FUNCTION_BLOCK EcMasterFrameCount IMPLEMENTS IEcTask
VAR_INPUT
END_VAR
VAR_OUTPUT
END_VAR
VAR
	iState : INT;
	masterFrameCount : Tc2_EtherCAT.FB_EcMasterFrameCount;
	_execute: BOOL;
	_done: BOOL;
	_busy: BOOL;
	_error: BOOL;
	_netId: AMSNETID;
END_VAR

CASE iState OF
	0:
		IF _execute THEN
			_done := FALSE;
			_busy := TRUE;
			_error := FALSE;
			masterFrameCount.bExecute := TRUE;
			IF masterFrameCount.bBusy THEN
				iState := 10;
				_execute := false;
			END_IF
		END_IF
	10:
		IF NOT masterFrameCount.bBusy THEN
			IF NOT masterFrameCount.bError THEN
				_done := TRUE;
			ELSE
				_error := TRUE;
			END_IF
			_busy := FALSE;
			masterFrameCount.bExecute := FALSE;
			iState := 0;
		END_IF
END_CASE

masterFrameCount(sNetId := Tc2_System.F_CreateAmsNetId(nIds := NetId));

{warning 'add method implementation '}
METHOD Abort : BOOL
masterFrameCount.bExecute := FALSE;
_busy := FALSE;
_execute := FALSE;
Abort := TRUE;
iState := 0;
END_METHOD

{warning 'add property implementation'}
PROPERTY Busy : BOOL
GET
Busy := _busy;
END_GET
END_PROPERTY

{warning 'add property implementation'}
PROPERTY Done : BOOL
GET
Done := _done;
END_GET
END_PROPERTY

{warning 'add property implementation'}
PROPERTY Error : BOOL
GET
Error := _error;
END_GET
END_PROPERTY

{warning 'add method implementation '}
METHOD Execute : BOOL
IF NOT masterFrameCount.bBusy THEN
	Execute := _execute := True;
END_IF
END_METHOD

PROPERTY FrameNumber : UDINT
GET
FrameNumber := masterFrameCount.nFrames;
END_GET
END_PROPERTY

{warning 'add property implementation'}
PROPERTY NetID : amsnetid
GET
NetID := _netId;
END_GET
SET
_netId := NetID;
END_SET
END_PROPERTY

END_FUNCTION_BLOCK

(* stored: Version 1.1.0.1, ProductVersion 3.1.4024.11
   POU EcMasterFrameCount: Id {09a697d0-71d0-4f6f-825d-38ffff5f388e}, SpecialFunc None
   Method Abort: Id {179768aa-7ee5-4432-82cc-810ed053a4fd}
   Property Busy: Id {4bfe5642-a7d0-419f-802d-2bd3a9224c56}
   Get Get: Id {c52382f8-0c4b-4390-a4a9-09a6f79c4179}
   Property Done: Id {3f07a710-3d2b-4135-ad6e-83a189d921f7}
   Get Get: Id {ff8561af-359e-455f-a02e-e0802c8faf50}
   Property Error: Id {413ba544-2d3c-43a8-b0af-54c895f8b9d5}
   Get Get: Id {74b39f58-dbdf-4c83-a937-eef82c5c05f0}
   Method Execute: Id {26056fc7-fae5-424d-932e-bfcd5fef20bf}
   Property FrameNumber: Id {1e6cc324-b1e2-48fe-8bc3-cad1d8d6fcc2}
   Get Get: Id {b8642ee9-420d-4204-9f0b-64a05d48ab2c}
   Property NetID: Id {5fb037c1-f58d-429e-964d-eb51ee36ad6a}
   Get Get: Id {ff6245ce-7869-45f7-9aa3-7f8199871515}
   Set Set: Id {6b315a97-ec91-4486-94eb-6bc7d8cddc7e} *)
